KUKA KRL data list: TEST_FREQ.dat

&ACCESS RVP
&REL 9
&PARAM TEMPLATE = C:\KRC\Roboter\Template\ExpertVorgabe
&PARAM EDITMASK = *
DEFDAT  TEST_FREQ PUBLIC
REAL FREQVAL=10.0308647
ENDDAT
